  rq_init_comm_if_connected(9, "1")
  rq_init_comm_if_connected(2, "2")
  rq_init_comm_if_connected(3, "3")
  rq_init_comm_if_connected(4, "4")
  rq_print_connected_grippers()
  rq_gripper_communication_thread = run rq_gripper_communication()
  set_closed_norm(100.0, 1)
  set_open_norm(0.0, 1)
  set_closed_mm(0.0, 1)
  set_open_mm(50.0, 1)
  set_closed_norm(100.0, 2)
  set_open_norm(0.0, 2)
  set_closed_mm(0.0, 2)
  set_open_mm(50.0, 2)
  set_closed_norm(100.0, 3)
  set_open_norm(0.0, 3)
  set_closed_mm(0.0, 3)
  set_open_mm(50.0, 3)
  set_closed_norm(100.0, 4)
  set_open_norm(0.0, 4)
  set_closed_mm(0.0, 4)
  set_open_mm(50.0, 4)
  rq_current_limit_enabled = False
  while(not rq_gripper_communication_thread_started):
      sleep(0.008)
  end
  # end: URCap Installation Node
  def ExtractCoinBattery():
    $ 40 "ExtractCoinBattery" "noBreak"
    $ 41 "wp_CoinBatApp≔wp_origin"
    global wp_CoinBatApp=wp_origin
    $ 42 "wp_CoinBatApp[0] = -0.0328"
    wp_CoinBatApp[0] = -0.0328
    $ 43 "wp_CoinBatApp[1] = 0.1238 + 0.002"
    wp_CoinBatApp[1] = 0.1238 + 0.002
    $ 44 "wp_CoinBatApp[2] = 0.07"
    wp_CoinBatApp[2] = 0.07
    $ 45 "MoveL"
    $ 46 "wp_CoinBatApp" "breakAfter"
    movel(pose_trans(Fearure_2_2P_Of, wp_CoinBatApp), a=1.2, v=0.25)
    $ 47 "wp_CoinBatExt≔wp_CoinBatApp"
    global wp_CoinBatExt=wp_CoinBatApp
    $ 48 "wp_CoinBatExt[2] = 0.115"
    wp_CoinBatExt[2] = 0.115
    $ 49 "MoveL"
    $ 50 "wp_CoinBatExt" "breakAfter"
    movel(pose_trans(Fearure_2_2P_Of, wp_CoinBatExt), a=1.2, v=0.25)
    # begin: URCap Program Node
    #   Source: Robotiq_Copilot, 1.22.1.14215, Robotiq Inc.
    #   Type: Find Surface
    $ 51 "Find Surface"
    rq_ft_sensor_disconnected_check()
    rq_zero_sensor()
    sleep(0.1)
    surface_found = rq_linear_search_urcap("X-", 35.000, 0.005000, 0.020000, 1)
    storevar.setvariablepose("rq_findSurface_d2ed8732-a4f1-4f80-aeeb-8b3bdc1d8fba_exitPosition", get_actual_tcp_pose())
    $ 52 "'Add Stop conditions from the Find Surface node'" "noBreak"
    # 'Add Stop conditions from the Find Surface node'
    # end: URCap Program Node
    $ 53 "Wait: 0"
    $ 54 "wp_CoinBatExt[2] = 0.07"
    wp_CoinBatExt[2] = 0.07
    $ 55 "MoveL"
    $ 56 "wp_CoinBatExt" "breakAfter"
    movel(pose_trans(Fearure_2_2P_Of, wp_CoinBatExt), a=1.2, v=0.25)
  end
  def PickPlaceCoinBattery():
    $ 59 "PickPlaceCoinBattery" "noBreak"
    # begin: URCap Program Node
    #   Source: Robotiq_Grippers, 1.8.8.13523, Robotiq Inc.
    #   Type: Gripper
    $ 60 "Gripper Move50% (1)"
    if not(gripper_connected[0]):
      popup("Gripper 1 must be connected to run this program.", "No connection", False, True, True)
    end
    if not(rq_is_gripper_activated("1")):
      popup("Gripper 1 is not activated. Go to Installation tab > Gripper to activate it and run the program again.", "Not activated", False, True, True)
    end
    rq_set_pos_spd_for(128, 255, 0, "1")
    rq_wait_pos_spe_for_request(128, 255, 0, "1")
    rq_go_to("1")
    rq_wait("1")
    # end: URCap Program Node
    $ 61 "wp_PickCoinApp≔wp_origin"
    global wp_PickCoinApp=wp_origin
    $ 62 "wp_PickCoinApp[0] = -0.0328"
    wp_PickCoinApp[0] = -0.0328
    $ 63 "wp_PickCoinApp[1] = 0.1238"
    wp_PickCoinApp[1] = 0.1238
    $ 64 "wp_PickCoinApp[2] = 0.14"
    wp_PickCoinApp[2] = 0.14
    $ 65 "wp_PickCoinApp[5] = d2r(90)"
    wp_PickCoinApp[5] = d2r(90)
    $ 66 "MoveL"
    $ 67 "wp_PickCoinApp" "breakAfter"
    movel(pose_trans(Fearure_2_2P_Of, wp_PickCoinApp), a=1.2, v=0.25)
    # begin: URCap Program Node
    #   Source: Robotiq_Grippers, 1.8.8.13523, Robotiq Inc.
    #   Type: Gripper
    $ 68 "Gripper Close (1)"
    if not(gripper_connected[0]):
      popup("Gripper 1 must be connected to run this program.", "No connection", False, True, True)
    end
    if not(rq_is_gripper_activated("1")):
      popup("Gripper 1 is not activated. Go to Installation tab > Gripper to activate it and run the program again.", "Not activated", False, True, True)
    end
    rq_set_pos_spd_for(255, 0, 0, "1")
    rq_wait_pos_spe_for_request(255, 0, 0, "1")
    rq_go_to("1")
    rq_wait("1")
    # end: URCap Program Node
    $ 69 "wp_PickCoinApp[2] = 0.12"
    wp_PickCoinApp[2] = 0.12
    $ 70 "MoveL"
    $ 71 "wp_PickCoinApp" "breakAfter"
    movel(pose_trans(Fearure_2_2P_Of, wp_PickCoinApp), a=1.2, v=0.25)
    $ 72 "wp_PickCoinApp[1] = 0.09"
    wp_PickCoinApp[1] = 0.09
    $ 73 "MoveL"
    $ 74 "wp_PickCoinApp" "breakAfter"
    movel(pose_trans(Fearure_2_2P_Of, wp_PickCoinApp), a=1.2, v=0.25)
    $ 75 "wp_PickCoinApp[2] = 0.13"
    wp_PickCoinApp[2] = 0.13
    $ 76 "MoveL"
    $ 77 "wp_PickCoinApp" "breakAfter"
    movel(pose_trans(Fearure_2_2P_Of, wp_PickCoinApp), a=1.2, v=0.25)
    # begin: URCap Program Node
    #   Source: Robotiq_Grippers, 1.8.8.13523, Robotiq Inc.
    #   Type: Gripper
    $ 78 "Gripper Move65% (1)"
    if not(gripper_connected[0]):
      popup("Gripper 1 must be connected to run this program.", "No connection", False, True, True)
    end
    if not(rq_is_gripper_activated("1")):
      popup("Gripper 1 is not activated. Go to Installation tab > Gripper to activate it and run the program again.", "Not activated", False, True, True)
    end
    rq_set_pos_spd_for(166, 0, 0, "1")
    rq_wait_pos_spe_for_request(166, 0, 0, "1")
    rq_go_to("1")
    rq_wait("1")
    # end: URCap Program Node
    $ 79 "wp_PickCoinApp[2] = 0"
    wp_PickCoinApp[2] = 0
    $ 80 "MoveL"
    $ 81 "wp_PickCoinApp" "breakAfter"
    movel(pose_trans(Fearure_2_2P_Of, wp_PickCoinApp), a=1.2, v=0.25)
    # begin: URCap Program Node
    #   Source: Robotiq_Grippers, 1.8.8.13523, Robotiq Inc.
    #   Type: Gripper
    $ 82 "Gripper Close (1)"
    if not(gripper_connected[0]):
      popup("Gripper 1 must be connected to run this program.", "No connection", False, True, True)
    end
    if not(rq_is_gripper_activated("1")):
      popup("Gripper 1 is not activated. Go to Installation tab > Gripper to activate it and run the program again.", "Not activated", False, True, True)
    end
    rq_set_pos_spd_for(255, 255, 0, "1")
    rq_wait_pos_spe_for_request(255, 255, 0, "1")
    rq_go_to("1")
    rq_wait("1")
    # end: URCap Program Node
  end
  def ExtractBattery2():
    $ 83 "ExtractBattery2" "noBreak"
    $ 84 "wp_Bat2ExtApp≔wp_origin"
    global wp_Bat2ExtApp=wp_origin
    $ 85 "wp_Bat2ExtApp[0] = -0.10"
    wp_Bat2ExtApp[0] = -0.10
    $ 86 "wp_Bat2ExtApp[1] = 0.06"
    wp_Bat2ExtApp[1] = 0.06
    $ 87 "wp_Bat2ExtApp[2] = 0.07"
    wp_Bat2ExtApp[2] = 0.07
    $ 88 "MoveL"
    $ 89 "wp_Bat2ExtApp" "breakAfter"
    movel(pose_trans(Fearure_2_2P_Of, wp_Bat2ExtApp), a=1.2, v=0.25)
    $ 90 "wp_Bat2ExtApp[2] = 0.115"
    wp_Bat2ExtApp[2] = 0.115
    $ 91 "MoveL"
    $ 92 "wp_Bat2ExtApp" "breakAfter"
    movel(pose_trans(Fearure_2_2P_Of, wp_Bat2ExtApp), a=1.2, v=0.25)
    # begin: URCap Program Node
    #   Source: Robotiq_Copilot, 1.22.1.14215, Robotiq Inc.
    #   Type: Find Surface
    $ 93 "Find Surface"
    rq_ft_sensor_disconnected_check()
    rq_zero_sensor()
    sleep(0.1)
    surface_found = rq_linear_search_urcap("X-", 30.000, 0.020000, 0.030000, 1)
    storevar.setvariablepose("rq_findSurface_fb726c3e-57f5-4e83-bd0d-2e451a65e373_exitPosition", get_actual_tcp_pose())
    $ 94 "'Add Stop conditions from the Find Surface node'" "noBreak"
    # 'Add Stop conditions from the Find Surface node'
    # end: URCap Program Node
    $ 95 "wp_Bat2ExtApp[2] = 0.07"
    wp_Bat2ExtApp[2] = 0.07
    $ 96 "MoveL"
    $ 97 "wp_Bat2ExtApp" "breakAfter"
    movel(pose_trans(Fearure_2_2P_Of, wp_Bat2ExtApp), a=1.2, v=0.25)
  end
  def PickTool():
    $ 98 "PickTool" "noBreak"
    $ 99 "wp_PickToolApp≔wp_CornerOrigin"
    global wp_PickToolApp=wp_CornerOrigin
    $ 100 "wp_PickToolApp[0] = -0.081"
    wp_PickToolApp[0] = -0.081
    $ 101 "wp_PickToolApp[1] = 0.083"
    wp_PickToolApp[1] = 0.083
    $ 102 "MoveL"
    $ 103 "wp_PickToolApp" "breakAfter"
    movel(pose_trans(Fearure_2_2P_Of, wp_PickToolApp), a=1.2, v=0.25)
    # begin: URCap Program Node
    #   Source: Robotiq_Grippers, 1.8.8.13523, Robotiq Inc.
    #   Type: Gripper
    $ 104 "Gripper Move60% (1)"
    if not(gripper_connected[0]):
      popup("Gripper 1 must be connected to run this program.", "No connection", False, True, True)
    end
    if not(rq_is_gripper_activated("1")):
      popup("Gripper 1 is not activated. Go to Installation tab > Gripper to activate it and run the program again.", "Not activated", False, True, True)
    end
    rq_set_pos_spd_for(153, 255, 0, "1")
    rq_wait_pos_spe_for_request(153, 255, 0, "1")
    rq_go_to("1")
    rq_wait("1")
    # end: URCap Program Node
    $ 105 "wp_PickToolApp[2] = 0.148"
    wp_PickToolApp[2] = 0.148
    $ 106 "MoveL"
    $ 107 "wp_PickToolApp" "breakAfter"
    movel(pose_trans(Fearure_2_2P_Of, wp_PickToolApp), a=1.2, v=0.25)
    $ 108 "wp_PickToolApp[1] = 0.08"
    wp_PickToolApp[1] = 0.08
    $ 109 "MoveL"
    $ 110 "wp_PickToolApp" "breakAfter"
    movel(pose_trans(Fearure_2_2P_Of, wp_PickToolApp), a=1.2, v=0.25)
    # begin: URCap Program Node
    #   Source: Robotiq_Grippers, 1.8.8.13523, Robotiq Inc.
    #   Type: Gripper
    $ 111 "Gripper Close (1)"
    if not(gripper_connected[0]):
      popup("Gripper 1 must be connected to run this program.", "No connection", False, True, True)
    end
    if not(rq_is_gripper_activated("1")):
      popup("Gripper 1 is not activated. Go to Installation tab > Gripper to activate it and run the program again.", "Not activated", False, True, True)
    end
    rq_set_pos_spd_for(255, 255, 255, "1")
    rq_wait_pos_spe_for_request(255, 255, 255, "1")
    rq_go_to("1")
    rq_wait("1")
    # end: URCap Program Node
    $ 112 "wp_PickToolApp[2] = 0.07"
    wp_PickToolApp[2] = 0.07
    $ 113 "MoveL"
    $ 114 "wp_PickToolApp" "breakAfter"
    movel(pose_trans(Fearure_2_2P_Of, wp_PickToolApp), a=1.2, v=0.25)
  end
  def PlaceTool():
    $ 115 "PlaceTool" "noBreak"
    $ 116 "wp_PlaceToolApp≔wp_origin"
    global wp_PlaceToolApp=wp_origin
    $ 117 "wp_PlaceToolApp[0] = -0.081"
    wp_PlaceToolApp[0] = -0.081
    $ 118 "wp_PlaceToolApp[1] = 0.08"
    wp_PlaceToolApp[1] = 0.08
    $ 119 "MoveL"
    $ 120 "wp_PlaceToolApp" "breakAfter"
    movel(pose_trans(Fearure_2_2P_Of, wp_PlaceToolApp), a=1.2, v=0.25)
    $ 121 "wp_PlaceToolApp[2] = 0.13"
    wp_PlaceToolApp[2] = 0.13
    $ 122 "MoveL"
    $ 123 "wp_PlaceToolApp" "breakAfter"
    movel(pose_trans(Fearure_2_2P_Of, wp_PlaceToolApp), a=1.2, v=0.25)
    # begin: URCap Program Node
    #   Source: Robotiq_Copilot, 1.22.1.14215, Robotiq Inc.
    #   Type: Insertion
    $ 124 "Insertion"
    rq_ft_sensor_disconnected_check()
    # begin: URCap Program Node
    #   Source: Robotiq_Copilot, 1.22.1.14215, Robotiq Inc.
    #   Type: Zero FT Sensor
    $ 125 "Zero FT Sensor" "noBreak"
    rq_ft_sensor_disconnected_check()
    rq_zero_sensor()
    # end: URCap Program Node
    # begin: URCap Program Node
    #   Source: Robotiq_Copilot, 1.22.1.14215, Robotiq Inc.
    #   Type: Linear
    $ 126 "Linear" "noBreak"
    rq_ft_sensor_disconnected_check()
    surface_found = rq_linear_search_urcap("Z+", 10.000, 0.020, 0.030, 1)
    # begin: URCap Program Node
    #   Source: Robotiq_Copilot, 1.22.1.14215, Robotiq Inc.
    #   Type: On error
    $ 127 "On error" "noBreak"
    if not(surface_found):
      $ 128 "'Sequence if maximum distance is reached'" "noBreak"
      # 'Sequence if maximum distance is reached'
      $ 129 "Halt" "noBreak"
      halt
    end
    # end: URCap Program Node
    # end: URCap Program Node
    # end: URCap Program Node
    # begin: URCap Program Node
    #   Source: Robotiq_Grippers, 1.8.8.13523, Robotiq Inc.
    #   Type: Gripper
    $ 130 "Gripper Move60% (1)"
    if not(gripper_connected[0]):
      popup("Gripper 1 must be connected to run this program.", "No connection", False, True, True)
    end
    if not(rq_is_gripper_activated("1")):
      popup("Gripper 1 is not activated. Go to Installation tab > Gripper to activate it and run the program again.", "Not activated", False, True, True)
    end
    rq_set_pos_spd_for(153, 255, 0, "1")
    rq_wait_pos_spe_for_request(153, 255, 0, "1")
    rq_go_to("1")
    rq_wait("1")
    # end: URCap Program Node
    $ 131 "wp_PlaceToolApp[2] = 0.07"
    wp_PlaceToolApp[2] = 0.07
    $ 132 "MoveL"
    $ 133 "wp_PlaceToolApp" "breakAfter"
    movel(pose_trans(Fearure_2_2P_Of, wp_PlaceToolApp), a=1.2, v=0.25)
    $ 134 "wp_PlaceToolApp[5] = 1.571"
    wp_PlaceToolApp[5] = 1.571
    $ 135 "MoveL"
    $ 136 "wp_PlaceToolApp" "breakAfter"
    movel(pose_trans(Fearure_2_2P_Of, wp_PlaceToolApp), a=1.2, v=0.25)
  end
  def ReleaseTool():
    $ 137 "ReleaseTool" "noBreak"
    $ 138 "wp_RelToolApp≔wp_origin"
    global wp_RelToolApp=wp_origin
    $ 139 "wp_RelToolApp[0] = -0.0328"
    wp_RelToolApp[0] = -0.0328
    $ 140 "wp_RelToolApp[1] = 0.18"
    wp_RelToolApp[1] = 0.18
    $ 141 "wp_RelToolApp[2] = 0.07"
    wp_RelToolApp[2] = 0.07
    $ 142 "MoveL"
    $ 143 "wp_RelToolApp" "breakAfter"
    movel(pose_trans(Fearure_2_2P_Of, wp_RelToolApp), a=1.2, v=0.25)
    # begin: URCap Program Node
    #   Source: Robotiq_Grippers, 1.8.8.13523, Robotiq Inc.
    #   Type: Gripper
    $ 144 "Gripper Move50% (1)"
    if not(gripper_connected[0]):
      popup("Gripper 1 must be connected to run this program.", "No connection", False, True, True)
    end
    if not(rq_is_gripper_activated("1")):
      popup("Gripper 1 is not activated. Go to Installation tab > Gripper to activate it and run the program again.", "Not activated", False, True, True)
    end
    rq_set_pos_spd_for(128, 255, 0, "1")
    rq_wait_pos_spe_for_request(128, 255, 0, "1")
    rq_go_to("1")
    rq_wait("1")
    # end: URCap Program Node
    $ 145 "wp_RelToolApp[2] = 0"
    wp_RelToolApp[2] = 0
    $ 146 "MoveL"
    $ 147 "wp_RelToolApp" "breakAfter"
    movel(pose_trans(Fearure_2_2P_Of, wp_RelToolApp), a=1.2, v=0.25)
    # begin: URCap Program Node
    #   Source: Robotiq_Grippers, 1.8.8.13523, Robotiq Inc.
    #   Type: Gripper
    $ 148 "Gripper Close (1)"
    if not(gripper_connected[0]):
      popup("Gripper 1 must be connected to run this program.", "No connection", False, True, True)
    end
    if not(rq_is_gripper_activated("1")):
      popup("Gripper 1 is not activated. Go to Installation tab > Gripper to activate it and run the program again.", "Not activated", False, True, True)
    end
    rq_set_pos_spd_for(255, 255, 0, "1")
    rq_wait_pos_spe_for_request(255, 255, 0, "1")
    rq_go_to("1")
    rq_wait("1")
    # end: URCap Program Node
  end
  def InsertBattery1():
    $ 149 "InsertBattery1" "noBreak"
    $ 150 "wp_InsBat1App≔wp_origin"
    global wp_InsBat1App=wp_origin
    $ 151 "wp_InsBat1App[0] = wp_InsBat1App[0] - 0.042"
    wp_InsBat1App[0] = wp_InsBat1App[0] - 0.042
    $ 152 "wp_InsBat1App[1] = wp_InsBat1App[1] + 0.0555"
    wp_InsBat1App[1] = wp_InsBat1App[1] + 0.0555
    $ 153 "MoveL"
    $ 154 "wp_InsBat1App" "breakAfter"
    movel(pose_trans(Fearure_2_2P_Of, wp_InsBat1App), a=1.2, v=0.25)
    $ 156 "wp_InsBat1App[2] = wp_InsBat1App[2] + 0.08"
    wp_InsBat1App[2] = wp_InsBat1App[2] + 0.08
    $ 157 "wp_InsBat1App[0] = wp_InsBat1App[0] + 0.005"
    wp_InsBat1App[0] = wp_InsBat1App[0] + 0.005
    $ 158 "MoveL"
    $ 159 "wp_InsBat1App" "breakAfter"
    movel(pose_trans(Fearure_2_2P_Of, wp_InsBat1App), a=1.2, v=0.25)
    # begin: URCap Program Node
    #   Source: Robotiq_Copilot, 1.22.1.14215, Robotiq Inc.
    #   Type: Insertion
    $ 160 "Insertion"
    rq_ft_sensor_disconnected_check()
    # begin: URCap Program Node
    #   Source: Robotiq_Copilot, 1.22.1.14215, Robotiq Inc.
    #   Type: Zero FT Sensor
    $ 161 "Zero FT Sensor" "noBreak"
    rq_ft_sensor_disconnected_check()
    rq_zero_sensor()
    # end: URCap Program Node
    # begin: URCap Program Node
    #   Source: Robotiq_Copilot, 1.22.1.14215, Robotiq Inc.
    #   Type: Linear
    $ 162 "Linear" "noBreak"
    rq_ft_sensor_disconnected_check()
    surface_found = rq_linear_search_urcap("Z+", 10.000, 0.010, 0.030, 1)
    # begin: URCap Program Node
    #   Source: Robotiq_Copilot, 1.22.1.14215, Robotiq Inc.
    #   Type: On error
    $ 163 "On error" "noBreak"
    if not(surface_found):
      $ 164 "'Sequence if maximum distance is reached'" "noBreak"
      # 'Sequence if maximum distance is reached'
      $ 165 "Halt" "noBreak"
      halt
    end
    # end: URCap Program Node
    # end: URCap Program Node
    # end: URCap Program Node
    $ 166 "Wait: 0.5"
    sleep(0.5)
    # begin: URCap Program Node
    #   Source: Robotiq_Grippers, 1.8.8.13523, Robotiq Inc.
    #   Type: Gripper
    $ 167 "Gripper Move60% (1)"
    if not(gripper_connected[0]):
      popup("Gripper 1 must be connected to run this program.", "No connection", False, True, True)
    end
    if not(rq_is_gripper_activated("1")):
      popup("Gripper 1 is not activated. Go to Installation tab > Gripper to activate it and run the program again.", "Not activated", False, True, True)
    end
    rq_set_pos_spd_for(153, 255, 0, "1")
    rq_wait_pos_spe_for_request(153, 255, 0, "1")
    rq_go_to("1")
    rq_wait("1")
    # end: URCap Program Node
    $ 168 "wp_InsBat1Ret≔wp_InsBat1App"
    global wp_InsBat1Ret=wp_InsBat1App
    $ 169 "wp_InsBat1Ret[2] = wp_InsBat1Ret[2] - 0.10"
    wp_InsBat1Ret[2] = wp_InsBat1Ret[2] - 0.10
    $ 170 "MoveL"
    $ 171 "wp_InsBat1Ret" "breakAfter"
    movel(pose_trans(Fearure_2_2P_Of, wp_InsBat1Ret), a=1.2, v=0.25)
    # begin: URCap Program Node
    #   Source: Robotiq_Grippers, 1.8.8.13523, Robotiq Inc.
    #   Type: Gripper
    $ 172 "Gripper Close (1)"
    if not(gripper_connected[0]):
      popup("Gripper 1 must be connected to run this program.", "No connection", False, True, True)
    end
    if not(rq_is_gripper_activated("1")):
      popup("Gripper 1 is not activated. Go to Installation tab > Gripper to activate it and run the program again.", "Not activated", False, True, True)
    end
    rq_set_pos_spd_for(255, 255, 0, "1")
    rq_wait_pos_spe_for_request(255, 255, 0, "1")
    rq_go_to("1")
    rq_wait("1")
    # end: URCap Program Node
  end
  def InsertBattery2():
    $ 179 "InsertBattery2" "noBreak"
    $ 180 "wp_InsBat2App≔wp_origin"
    global wp_InsBat2App=wp_origin
    $ 181 "wp_InsBat2App[0] = -0.058"
    wp_InsBat2App[0] = -0.058
    $ 182 "wp_InsBat2App[1] = 0.0555"
    wp_InsBat2App[1] = 0.0555
    $ 183 "wp_InsBat2App[5] = 1.571"
    wp_InsBat2App[5] = 1.571
    $ 184 "MoveL"
    $ 185 "wp_InsBat2App" "breakAfter"
    movel(pose_trans(Fearure_2_2P_Of, wp_InsBat2App), a=1.2, v=0.25)
    $ 186 "wp_InsBat2App[2] = 0.08"
    wp_InsBat2App[2] = 0.08
    $ 187 "wp_InsBat2App[0] = wp_InsBat2App[0] - 0.005"
    wp_InsBat2App[0] = wp_InsBat2App[0] - 0.005
    $ 188 "MoveL"
    $ 189 "wp_InsBat2App" "breakAfter"
    movel(pose_trans(Fearure_2_2P_Of, wp_InsBat2App), a=1.2, v=0.25)
    # begin: URCap Program Node
    #   Source: Robotiq_Copilot, 1.22.1.14215, Robotiq Inc.
    #   Type: Insertion
    $ 190 "Insertion"
    rq_ft_sensor_disconnected_check()
    # begin: URCap Program Node
    #   Source: Robotiq_Copilot, 1.22.1.14215, Robotiq Inc.
    #   Type: Zero FT Sensor
    $ 191 "Zero FT Sensor" "noBreak"
    rq_ft_sensor_disconnected_check()
    rq_zero_sensor()
    # end: URCap Program Node
    # begin: URCap Program Node
    #   Source: Robotiq_Copilot, 1.22.1.14215, Robotiq Inc.
    #   Type: Linear
    $ 192 "Linear" "noBreak"
    rq_ft_sensor_disconnected_check()
    surface_found = rq_linear_search_urcap("Z+", 10.000, 0.010, 0.030, 1)
    # begin: URCap Program Node
    #   Source: Robotiq_Copilot, 1.22.1.14215, Robotiq Inc.
    #   Type: On error
    $ 193 "On error" "noBreak"
    if not(surface_found):
      $ 194 "'Sequence if maximum distance is reached'" "noBreak"
      # 'Sequence if maximum distance is reached'
      $ 195 "Halt" "noBreak"
      halt
    end
    # end: URCap Program Node
    # end: URCap Program Node
    # end: URCap Program Node
    $ 196 "Wait: 0.5"
    sleep(0.5)
    # begin: URCap Program Node
    #   Source: Robotiq_Grippers, 1.8.8.13523, Robotiq Inc.
    #   Type: Gripper
    $ 197 "Gripper Move60% (1)"
    if not(gripper_connected[0]):
      popup("Gripper 1 must be connected to run this program.", "No connection", False, True, True)
    end
    if not(rq_is_gripper_activated("1")):
      popup("Gripper 1 is not activated. Go to Installation tab > Gripper to activate it and run the program again.", "Not activated", False, True, True)
    end
    rq_set_pos_spd_for(153, 255, 0, "1")
    rq_wait_pos_spe_for_request(153, 255, 0, "1")
    rq_go_to("1")
    rq_wait("1")
    # end: URCap Program Node
    $ 198 "wp_InsBat2Ret≔wp_InsBat2App"
    global wp_InsBat2Ret=wp_InsBat2App
    $ 199 "wp_InsBat2Ret[2] = wp_InsBat2Ret[2] - 0.10"
    wp_InsBat2Ret[2] = wp_InsBat2Ret[2] - 0.10
    $ 200 "MoveL"
    $ 201 "wp_InsBat2Ret" "breakAfter"
    movel(pose_trans(Fearure_2_2P_Of, wp_InsBat2Ret), a=1.2, v=0.25)
    # begin: URCap Program Node
    #   Source: Robotiq_Grippers, 1.8.8.13523, Robotiq Inc.
    #   Type: Gripper
    $ 202 "Gripper Close (1)"
    if not(gripper_connected[0]):
      popup("Gripper 1 must be connected to run this program.", "No connection", False, True, True)
    end
    if not(rq_is_gripper_activated("1")):
      popup("Gripper 1 is not activated. Go to Installation tab > Gripper to activate it and run the program again.", "Not activated", False, True, True)
    end
    rq_set_pos_spd_for(255, 255, 0, "1")
    rq_wait_pos_spe_for_request(255, 255, 0, "1")
    rq_go_to("1")
    rq_wait("1")
    # end: URCap Program Node
  end
  def PickBattery2():
    $ 203 "PickBattery2" "noBreak"
    # begin: URCap Program Node
    #   Source: Robotiq_Grippers, 1.8.8.13523, Robotiq Inc.
    #   Type: Gripper
    $ 204 "Gripper Move60% (1)"
    if not(gripper_connected[0]):
      popup("Gripper 1 must be connected to run this program.", "No connection", False, True, True)
    end
    if not(rq_is_gripper_activated("1")):
      popup("Gripper 1 is not activated. Go to Installation tab > Gripper to activate it and run the program again.", "Not activated", False, True, True)
    end
    rq_set_pos_spd_for(153, 0, 0, "1")
    rq_wait_pos_spe_for_request(153, 0, 0, "1")
    rq_go_to("1")
    rq_wait("1")
    # end: URCap Program Node
    $ 205 "wp_Bat2PickApp≔wp_origin"
    global wp_Bat2PickApp=wp_origin
    $ 206 "wp_Bat2PickApp[0] = -0.1045"
    wp_Bat2PickApp[0] = -0.1045
    $ 207 "wp_Bat2PickApp[1] = 0.0565"
    wp_Bat2PickApp[1] = 0.0565
    $ 208 "wp_Bat2PickApp[5] = 1.571"
    wp_Bat2PickApp[5] = 1.571
    $ 209 "MoveL"
    $ 210 "wp_Bat2PickApp" "breakAfter"
    movel(pose_trans(Fearure_2_2P_Of, wp_Bat2PickApp), a=1.2, v=0.25)
    $ 211 "wp_Bat2PickApp[2] = 0.134"
    wp_Bat2PickApp[2] = 0.134
    $ 212 "MoveL"
    $ 213 "wp_Bat2PickApp" "breakAfter"
    movel(pose_trans(Fearure_2_2P_Of, wp_Bat2PickApp), a=1.2, v=0.25)
    # begin: URCap Program Node
    #   Source: Robotiq_Grippers, 1.8.8.13523, Robotiq Inc.
    #   Type: Gripper
    $ 214 "Gripper Close (1)"
    if not(gripper_connected[0]):
      popup("Gripper 1 must be connected to run this program.", "No connection", False, True, True)
    end
    if not(rq_is_gripper_activated("1")):
      popup("Gripper 1 is not activated. Go to Installation tab > Gripper to activate it and run the program again.", "Not activated", False, True, True)
    end
    rq_set_pos_spd_for(255, 128, 0, "1")
    rq_wait_pos_spe_for_request(255, 128, 0, "1")
    rq_go_to("1")
    rq_wait("1")
    # end: URCap Program Node
    $ 215 "wp_Bat2PickApp[2] = 0.07"
    wp_Bat2PickApp[2] = 0.07
    $ 216 "MoveL"
    $ 217 "wp_Bat2PickApp" "breakAfter"
    movel(pose_trans(Fearure_2_2P_Of, wp_Bat2PickApp), a=1.2, v=0.25)
    # begin: URCap Program Node
    #   Source: Robotiq_Grippers, 1.8.8.13523, Robotiq Inc.
    #   Type: Gripper
    $ 218 "Gripper Move72% (1)"
    if not(gripper_connected[0]):
      popup("Gripper 1 must be connected to run this program.", "No connection", False, True, True)
    end
    if not(rq_is_gripper_activated("1")):
      popup("Gripper 1 is not activated. Go to Installation tab > Gripper to activate it and run the program again.", "Not activated", False, True, True)
    end
    rq_set_pos_spd_for(184, 0, 0, "1")
    rq_wait_pos_spe_for_request(184, 0, 0, "1")
    rq_go_to("1")
    rq_wait("1")
    # end: URCap Program Node
    $ 219 "Wait: 3.0"
    sleep(3.0)
    # begin: URCap Program Node
    #   Source: Robotiq_Grippers, 1.8.8.13523, Robotiq Inc.
    #   Type: Gripper
    $ 220 "Gripper Move85% (1)"
    if not(gripper_connected[0]):
      popup("Gripper 1 must be connected to run this program.", "No connection", False, True, True)
    end
    if not(rq_is_gripper_activated("1")):
      popup("Gripper 1 is not activated. Go to Installation tab > Gripper to activate it and run the program again.", "Not activated", False, True, True)
    end
    rq_set_pos_spd_for(217, 255, 0, "1")
    rq_wait_pos_spe_for_request(217, 255, 0, "1")
    rq_go_to("1")
    rq_wait("1")
    # end: URCap Program Node
  end
  def PickBattery1():
    $ 221 "PickBattery1" "noBreak"
    # begin: URCap Program Node
    #   Source: Robotiq_Grippers, 1.8.8.13523, Robotiq Inc.
    #   Type: Gripper
    $ 222 "Gripper Move60% (1)"
    if not(gripper_connected[0]):
      popup("Gripper 1 must be connected to run this program.", "No connection", False, True, True)
    end
    if not(rq_is_gripper_activated("1")):
      popup("Gripper 1 is not activated. Go to Installation tab > Gripper to activate it and run the program again.", "Not activated", False, True, True)
    end
    rq_set_pos_spd_for(153, 0, 0, "1")
    rq_wait_pos_spe_for_request(153, 0, 0, "1")
    rq_go_to("1")
    rq_wait("1")
    # end: URCap Program Node
    $ 223 "wp_Bat1ExtApp≔wp_origin"
    global wp_Bat1ExtApp=wp_origin
    $ 224 "wp_Bat1ExtApp[0] = wp_Bat1ExtApp[0] - 0.1540"
    wp_Bat1ExtApp[0] = wp_Bat1ExtApp[0] - 0.1540
    $ 225 "wp_Bat1ExtApp[1] = wp_Bat1ExtApp[1] + 0.0415"
    wp_Bat1ExtApp[1] = wp_Bat1ExtApp[1] + 0.0415
    $ 226 "wp_Bat1ExtApp[5] = wp_Bat1ExtApp[5] + 1.571"
    wp_Bat1ExtApp[5] = wp_Bat1ExtApp[5] + 1.571
    $ 227 "MoveL"
    $ 228 "wp_Bat1ExtApp" "breakAfter"
    movel(pose_trans(Fearure_2_2P_Of, wp_Bat1ExtApp), a=1.2, v=0.25)
    $ 229 "wp_Bat1ExtApp[2] = wp_Bat1ExtApp[2] + 0.136"
    wp_Bat1ExtApp[2] = wp_Bat1ExtApp[2] + 0.136
    $ 230 "MoveL"
    $ 231 "wp_Bat1ExtApp" "breakAfter"
    movel(pose_trans(Fearure_2_2P_Of, wp_Bat1ExtApp), a=1.2, v=0.25)
    # begin: URCap Program Node
    #   Source: Robotiq_Grippers, 1.8.8.13523, Robotiq Inc.
    #   Type: Gripper
    $ 232 "Gripper Close (1)"
    if not(gripper_connected[0]):
      popup("Gripper 1 must be connected to run this program.", "No connection", False, True, True)
    end
    if not(rq_is_gripper_activated("1")):
      popup("Gripper 1 is not activated. Go to Installation tab > Gripper to activate it and run the program again.", "Not activated", False, True, True)
    end
    rq_set_pos_spd_for(255, 0, 0, "1")
    rq_wait_pos_spe_for_request(255, 0, 0, "1")
    rq_go_to("1")
    rq_wait("1")
    # end: URCap Program Node
    $ 233 "wp_Bat1ExtApp[2] = wp_Bat1ExtApp[2] - 0.10"
    wp_Bat1ExtApp[2] = wp_Bat1ExtApp[2] - 0.10
    $ 234 "MoveL"
    $ 235 "wp_Bat1ExtApp" "breakAfter"
    movel(pose_trans(Fearure_2_2P_Of, wp_Bat1ExtApp), a=1.2, v=0.25)
    # begin: URCap Program Node
    #   Source: Robotiq_Grippers, 1.8.8.13523, Robotiq Inc.
    #   Type: Gripper
    $ 236 "Gripper Move72% (1)"
    if not(gripper_connected[0]):
      popup("Gripper 1 must be connected to run this program.", "No connection", False, True, True)
    end
    if not(rq_is_gripper_activated("1")):
      popup("Gripper 1 is not activated. Go to Installation tab > Gripper to activate it and run the program again.", "Not activated", False, True, True)
    end
    rq_set_pos_spd_for(184, 0, 0, "1")
    rq_wait_pos_spe_for_request(184, 0, 0, "1")
    rq_go_to("1")
    rq_wait("1")
    # end: URCap Program Node
    $ 237 "Wait: 3.0"
    sleep(3.0)
    # begin: URCap Program Node
    #   Source: Robotiq_Grippers, 1.8.8.13523, Robotiq Inc.
    #   Type: Gripper
    $ 238 "Gripper Move85% (1)"
    if not(gripper_connected[0]):
      popup("Gripper 1 must be connected to run this program.", "No connection", False, True, True)
    end
    if not(rq_is_gripper_activated("1")):
      popup("Gripper 1 is not activated. Go to Installation tab > Gripper to activate it and run the program again.", "Not activated", False, True, True)
    end
    rq_set_pos_spd_for(217, 255, 0, "1")
    rq_wait_pos_spe_for_request(217, 255, 0, "1")
    rq_go_to("1")
    rq_wait("1")
    # end: URCap Program Node
  end
  def ExtractBattery1():
    $ 239 "ExtractBattery1" "noBreak"
    $ 240 "wp_Bat1ExtApp≔wp_origin"
    global wp_Bat1ExtApp=wp_origin
    $ 241 "wp_Bat1ExtApp[0] = wp_Bat1ExtApp[0] - 0.1540"
    wp_Bat1ExtApp[0] = wp_Bat1ExtApp[0] - 0.1540
    $ 242 "wp_Bat1ExtApp[1] = wp_Bat1ExtApp[1] + 0.0415"
    wp_Bat1ExtApp[1] = wp_Bat1ExtApp[1] + 0.0415
    $ 243 "MoveL"
    $ 244 "wp_Bat1ExtApp" "breakAfter"
    movel(pose_trans(Fearure_2_2P_Of, wp_Bat1ExtApp), a=1.2, v=0.25)
    # begin: URCap Program Node
    #   Source: Robotiq_Grippers, 1.8.8.13523, Robotiq Inc.
    #   Type: Gripper
    $ 245 "Gripper Move30% (1)"
    if not(gripper_connected[0]):
      popup("Gripper 1 must be connected to run this program.", "No connection", False, True, True)
    end
    if not(rq_is_gripper_activated("1")):
      popup("Gripper 1 is not activated. Go to Installation tab > Gripper to activate it and run the program again.", "Not activated", False, True, True)
    end
    rq_set_pos_spd_for(77, 0, 0, "1")
    rq_wait_pos_spe_for_request(77, 0, 0, "1")
    rq_go_to("1")
    rq_wait("1")
    # end: URCap Program Node
    $ 246 "wp_Bat1Extract≔wp_Bat1ExtApp"
    global wp_Bat1Extract=wp_Bat1ExtApp
    $ 247 "wp_Bat1Extract[0] = wp_Bat1Extract[0] + 0.034"
    wp_Bat1Extract[0] = wp_Bat1Extract[0] + 0.034
    $ 248 "wp_Bat1Extract[1] = wp_Bat1Extract[1] - 0.01"
    wp_Bat1Extract[1] = wp_Bat1Extract[1] - 0.01
    $ 249 "wp_Bat1Extract[2] = wp_Bat1Extract[2] + 0.145"
    wp_Bat1Extract[2] = wp_Bat1Extract[2] + 0.145
    $ 250 "MoveL"
    $ 251 "wp_Bat1Extract" "breakAfter"
    movel(pose_trans(Fearure_2_2P_Of, wp_Bat1Extract), a=1.2, v=0.25)
    # begin: URCap Program Node
    #   Source: Robotiq_Copilot, 1.22.1.14215, Robotiq Inc.
    #   Type: Find Surface
    $ 252 "Find Surface"
    rq_ft_sensor_disconnected_check()
    rq_zero_sensor()
    sleep(0.1)
    surface_found = rq_linear_search_urcap("X+", 30.000, 0.030000, 0.010000, 1)
    storevar.setvariablepose("rq_findSurface_26ca67e9-cc0e-4d30-826d-8f6b0826683b_exitPosition", get_actual_tcp_pose())
    $ 253 "'Add Stop conditions from the Find Surface node'" "noBreak"
    # 'Add Stop conditions from the Find Surface node'
    # end: URCap Program Node
    $ 254 "wp_Bat1Extract[2] = wp_Bat1Extract[2] - 0.05"
    wp_Bat1Extract[2] = wp_Bat1Extract[2] - 0.05
    $ 255 "MoveL"
    $ 256 "wp_Bat1Extract" "breakAfter"
    movel(pose_trans(Fearure_2_2P_Of, wp_Bat1Extract), a=1.2, v=0.5)
    # begin: URCap Program Node
    #   Source: Robotiq_Grippers, 1.8.8.13523, Robotiq Inc.
    #   Type: Gripper
    $ 257 "Gripper Move60% (1)"
    if not(gripper_connected[0]):
      popup("Gripper 1 must be connected to run this program.", "No connection", False, True, True)
    end
    if not(rq_is_gripper_activated("1")):
      popup("Gripper 1 is not activated. Go to Installation tab > Gripper to activate it and run the program again.", "Not activated", False, True, True)
    end
    rq_set_pos_spd_for(153, 0, 0, "1")
    rq_wait_pos_spe_for_request(153, 0, 0, "1")
    rq_go_to("1")
    rq_wait("1")
    # end: URCap Program Node
  end
  def AABatteryCoverExtraction():
    $ 258 "AABatteryCoverExtraction" "noBreak"
    $ 259 "wp_AABatCovApp≔wp_origin"
    global wp_AABatCovApp=wp_origin
    $ 260 "wp_AABatCovApp[0] = wp_AABatCovApp[0] - 0.1125"
    wp_AABatCovApp[0] = wp_AABatCovApp[0] - 0.1125
    $ 261 "wp_AABatCovApp[1] = wp_AABatCovApp[1] + 0.0485"
    wp_AABatCovApp[1] = wp_AABatCovApp[1] + 0.0485
    $ 262 "MoveL"
    $ 263 "wp_AABatCovApp" "breakAfter"
    movel(pose_trans(Fearure_2_2P_Of, wp_AABatCovApp), a=1.2, v=0.25)
    $ 264 "wp_AABatCovPres≔wp_AABatCovApp"
    global wp_AABatCovPres=wp_AABatCovApp
    $ 265 "wp_AABatCovPres[3] = wp_AABatCovPres[3] + 0.7854"
    wp_AABatCovPres[3] = wp_AABatCovPres[3] + 0.7854
    $ 266 "wp_AABatCovPres[2] = wp_AABatCovPres[2] + 0.12"
    wp_AABatCovPres[2] = wp_AABatCovPres[2] + 0.12
    $ 267 "wp_AABatCovPres[1] = wp_AABatCovPres[1] - 0.008"
    wp_AABatCovPres[1] = wp_AABatCovPres[1] - 0.008
    $ 268 "wp_AABatCovPres[0] = wp_AABatCovPres[0] + 0.005"
    wp_AABatCovPres[0] = wp_AABatCovPres[0] + 0.005
    $ 269 "MoveL"
    $ 270 "wp_AABatCovPres" "breakAfter"
    movel(pose_trans(Fearure_2_2P_Of, wp_AABatCovPres), a=1.2, v=0.25)
    # begin: URCap Program Node
    #   Source: Robotiq_Copilot, 1.22.1.14215, Robotiq Inc.
    #   Type: Find Surface
    $ 271 "Find Surface"
    rq_ft_sensor_disconnected_check()
    rq_zero_sensor()
    sleep(0.1)
    surface_found = rq_linear_search_urcap("Z-", 15.000, 0.030000, 0.010000, 0)
    storevar.setvariablepose("rq_findSurface_54677085-d0b4-4075-8ce2-dc145cac5c67_exitPosition", get_actual_tcp_pose())
    $ 272 "'Add Stop conditions from the Find Surface node'" "noBreak"
    # 'Add Stop conditions from the Find Surface node'
    # end: URCap Program Node
    $ 273 "wp_AABatCovRem≔wp_AABatCovPres"
    global wp_AABatCovRem=wp_AABatCovPres
    $ 274 "wp_AABatCovRem[2] = wp_AABatCovRem[2] + 0.009"
    wp_AABatCovRem[2] = wp_AABatCovRem[2] + 0.009
    $ 275 "wp_AABatCovRem[0] = wp_AABatCovRem[0] - 0.07"
    wp_AABatCovRem[0] = wp_AABatCovRem[0] - 0.07
    $ 276 "MoveL"
    $ 277 "wp_AABatCovRem" "breakAfter"
    movel(pose_trans(Fearure_2_2P_Of, wp_AABatCovRem), a=1.2, v=0.25)
  end
  def PlugInsertion():
    $ 294 "PlugInsertion" "noBreak"
    $ 295 "wp_PlgInsApp≔wp_origin"
    global wp_PlgInsApp=wp_origin
    $ 296 "wp_PlgInsApp[0] =wp_PlgInsApp[0] - 0.1390"
    wp_PlgInsApp[0] =wp_PlgInsApp[0] - 0.1390
    $ 297 "wp_PlgInsApp[1] =wp_PlgInsApp[1] + 0.1065"
    wp_PlgInsApp[1] =wp_PlgInsApp[1] + 0.1065
    $ 298 "wp_PlgInsApp[2] =wp_PlgInsApp[2] + 0.1085"
    wp_PlgInsApp[2] =wp_PlgInsApp[2] + 0.1085
    $ 299 "wp_PlgInsApp[5] = 1.571"
    wp_PlgInsApp[5] = 1.571
    $ 300 "MoveL"
    $ 301 "wp_PlgInsApp" "breakAfter"
    movel(pose_trans(Fearure_2_2P_Of, wp_PlgInsApp), a=1.2, v=0.25)
    $ 302 "wp_PlgInsertion≔wp_PlgInsApp"
    global wp_PlgInsertion=wp_PlgInsApp
    $ 303 "wp_PlgInsertion[2] = wp_PlgInsertion[2] + 0.025"
    wp_PlgInsertion[2] = wp_PlgInsertion[2] + 0.025
    $ 304 "MoveL"
    $ 305 "wp_PlgInsertion" "breakAfter"
    movel(pose_trans(Fearure_2_2P_Of, wp_PlgInsertion), a=1.2, v=0.25)
    # begin: URCap Program Node
    #   Source: Robotiq_Copilot, 1.22.1.14215, Robotiq Inc.
    #   Type: Insertion
    $ 306 "Insertion"
    rq_ft_sensor_disconnected_check()
    # begin: URCap Program Node
    #   Source: Robotiq_Copilot, 1.22.1.14215, Robotiq Inc.
    #   Type: Zero FT Sensor
    $ 307 "Zero FT Sensor" "noBreak"
    rq_ft_sensor_disconnected_check()
    rq_zero_sensor()
    # end: URCap Program Node
    # begin: URCap Program Node
    #   Source: Robotiq_Copilot, 1.22.1.14215, Robotiq Inc.
    #   Type: Linear
    $ 308 "Linear" "noBreak"
    rq_ft_sensor_disconnected_check()
    surface_found = rq_linear_search_urcap("Z+", 10.000, 0.010, 0.015, 1)
    # begin: URCap Program Node
    #   Source: Robotiq_Copilot, 1.22.1.14215, Robotiq Inc.
    #   Type: On error
    $ 309 "On error" "noBreak"
    if not(surface_found):
      $ 310 "'Sequence if maximum distance is reached'" "noBreak"
      # 'Sequence if maximum distance is reached'
      $ 311 "Halt" "noBreak"
      halt
    end
    # end: URCap Program Node
    # end: URCap Program Node
    # end: URCap Program Node
    # begin: URCap Program Node
    #   Source: Robotiq_Grippers, 1.8.8.13523, Robotiq Inc.
    #   Type: Gripper
    $ 312 "Gripper Move60% (1)"
    if not(gripper_connected[0]):
      popup("Gripper 1 must be connected to run this program.", "No connection", False, True, True)
    end
    if not(rq_is_gripper_activated("1")):
      popup("Gripper 1 is not activated. Go to Installation tab > Gripper to activate it and run the program again.", "Not activated", False, True, True)
    end
    rq_set_pos_spd_for(153, 128, 0, "1")
    rq_wait_pos_spe_for_request(153, 128, 0, "1")
    rq_go_to("1")
    rq_wait("1")
    # end: URCap Program Node
    $ 313 "wp_PlgInsRet≔wp_PlgInsertion"
    global wp_PlgInsRet=wp_PlgInsertion
    $ 314 "wp_PlgInsRet[2] = wp_PlgInsRet[2] - 0.1485"
    wp_PlgInsRet[2] = wp_PlgInsRet[2] - 0.1485
    $ 315 "MoveL"
    $ 316 "wp_PlgInsRet" "breakAfter"
    movel(pose_trans(Fearure_2_2P_Of, wp_PlgInsRet), a=1.2, v=0.25)
    # begin: URCap Program Node
    #   Source: Robotiq_Grippers, 1.8.8.13523, Robotiq Inc.
    #   Type: Gripper
    $ 317 "Gripper Close (1)"
    if not(gripper_connected[0]):
      popup("Gripper 1 must be connected to run this program.", "No connection", False, True, True)
    end
    if not(rq_is_gripper_activated("1")):
      popup("Gripper 1 is not activated. Go to Installation tab > Gripper to activate it and run the program again.", "Not activated", False, True, True)
    end
    rq_set_pos_spd_for(255, 128, 0, "1")
    rq_wait_pos_spe_for_request(255, 128, 0, "1")
    rq_go_to("1")
    rq_wait("1")
    # end: URCap Program Node
    $ 318 "wp_PlgInsRet[5] = 0"
    wp_PlgInsRet[5] = 0
    $ 319 "MoveL"
    $ 320 "wp_PlgInsRet" "breakAfter"
    movel(pose_trans(Fearure_2_2P_Of, wp_PlgInsRet), a=1.2, v=0.25)
  end
  def PlugExtraction():
    $ 321 "PlugExtraction" "noBreak"
    $ 322 "wp_PlgExtApp≔wp_origin"
    global wp_PlgExtApp=wp_origin
    $ 323 "wp_PlgExtApp[0] = wp_PlgExtApp[0] - 0.0990"
    wp_PlgExtApp[0] = wp_PlgExtApp[0] - 0.0990
    $ 324 "wp_PlgExtApp[1] = wp_PlgExtApp[1] + 0.1075"
    wp_PlgExtApp[1] = wp_PlgExtApp[1] + 0.1075
    $ 325 "wp_PlgExtApp[5] = 1.571"
    wp_PlgExtApp[5] = 1.571
    $ 326 "MoveL"
    $ 327 "wp_PlgExtApp" "breakAfter"
    movel(pose_trans(Fearure_2_2P_Of, wp_PlgExtApp), a=1.2, v=0.25)
    # begin: URCap Program Node
    #   Source: Robotiq_Grippers, 1.8.8.13523, Robotiq Inc.
    #   Type: Gripper
    $ 328 "Gripper Move60% (1)"
    if not(gripper_connected[0]):
      popup("Gripper 1 must be connected to run this program.", "No connection", False, True, True)
    end
    if not(rq_is_gripper_activated("1")):
      popup("Gripper 1 is not activated. Go to Installation tab > Gripper to activate it and run the program again.", "Not activated", False, True, True)
    end
    rq_set_pos_spd_for(153, 0, 0, "1")
    rq_wait_pos_spe_for_request(153, 0, 0, "1")
    rq_go_to("1")
    rq_wait("1")
    # end: URCap Program Node
    $ 329 "wp_PlgExtract≔wp_PlgExtApp"
    global wp_PlgExtract=wp_PlgExtApp
    $ 330 "wp_PlgExtract[2] = wp_PlgExtract[2] + 0.1385"
    wp_PlgExtract[2] = wp_PlgExtract[2] + 0.1385
    $ 331 "MoveL"
    $ 332 "wp_PlgExtract" "breakAfter"
    movel(pose_trans(Fearure_2_2P_Of, wp_PlgExtract), a=1.2, v=0.25)
    # begin: URCap Program Node
    #   Source: Robotiq_Grippers, 1.8.8.13523, Robotiq Inc.
    #   Type: Gripper
    $ 333 "Gripper Close (1)"
    if not(gripper_connected[0]):
      popup("Gripper 1 must be connected to run this program.", "No connection", False, True, True)
    end
    if not(rq_is_gripper_activated("1")):
      popup("Gripper 1 is not activated. Go to Installation tab > Gripper to activate it and run the program again.", "Not activated", False, True, True)
    end
    rq_set_pos_spd_for(255, 0, 255, "1")
    rq_wait_pos_spe_for_request(255, 0, 255, "1")
    rq_go_to("1")
    rq_wait("1")
    # end: URCap Program Node
    $ 334 "wp_PlgExtRet≔wp_PlgExtract"
    global wp_PlgExtRet=wp_PlgExtract
    $ 335 "wp_PlgExtRet[2] = wp_PlgExtRet[2] - 0.03"
    wp_PlgExtRet[2] = wp_PlgExtRet[2] - 0.03
    $ 336 "MoveL"
    $ 337 "wp_PlgExtRet" "breakAfter"
    movel(pose_trans(Fearure_2_2P_Of, wp_PlgExtRet), a=1.2, v=0.25)
  end
  def KeyInsertion():
    $ 338 "KeyInsertion" "noBreak"
    $ 339 "wp_KeyInsApp≔wp_origin"
    global wp_KeyInsApp=wp_origin
    $ 340 "wp_KeyInsApp[0] = -0.1835 + 0.001"
    wp_KeyInsApp[0] = -0.1835 + 0.001
    $ 341 "wp_KeyInsApp[1] = 0.1105 - 0.003"
    wp_KeyInsApp[1] = 0.1105 - 0.003
    $ 342 "wp_KeyInsApp[5] = 0"
    wp_KeyInsApp[5] = 0
    $ 343 "MoveL"
    $ 344 "wp_KeyInsApp" "breakAfter"
    movel(pose_trans(Fearure_2_2P_Of, wp_KeyInsApp), a=1.2, v=0.25)
    $ 345 "wp_KeyInsert≔wp_KeyInsApp"
    global wp_KeyInsert=wp_KeyInsApp
    $ 346 "wp_KeyInsert[2] = 0.111"
    wp_KeyInsert[2] = 0.111
    $ 347 "MoveL"
    $ 348 "wp_KeyInsert" "breakAfter"
    movel(pose_trans(Fearure_2_2P_Of, wp_KeyInsert), a=1.2, v=0.25)
    # begin: URCap Program Node
    #   Source: Robotiq_Copilot, 1.22.1.14215, Robotiq Inc.
    #   Type: Insertion
    $ 349 "Insertion"
    rq_ft_sensor_disconnected_check()
    # begin: URCap Program Node
    #   Source: Robotiq_Copilot, 1.22.1.14215, Robotiq Inc.
    #   Type: Zero FT Sensor
    $ 350 "Zero FT Sensor" "noBreak"
    rq_ft_sensor_disconnected_check()
    rq_zero_sensor()
    # end: URCap Program Node
    # begin: URCap Program Node
    #   Source: Robotiq_Copilot, 1.22.1.14215, Robotiq Inc.
    #   Type: Linear
    $ 351 "Linear" "noBreak"
    rq_ft_sensor_disconnected_check()
    surface_found = rq_linear_search_urcap("Z+", 10.000, 0.020, 0.030, 1)
    # begin: URCap Program Node
    #   Source: Robotiq_Copilot, 1.22.1.14215, Robotiq Inc.
    #   Type: On error
    $ 352 "On error" "noBreak"
    if not(surface_found):
      $ 353 "'Sequence if maximum distance is reached'" "noBreak"
      # 'Sequence if maximum distance is reached'
      $ 354 "Halt" "noBreak"
      halt
    end
    # end: URCap Program Node
    # end: URCap Program Node
    # end: URCap Program Node
    $ 355 "KeyFeature = get_actual_tcp_pose()"
    KeyFeature =  get_actual_tcp_pose ()
    $ 356 "wp_KeyOrigin[5] = d2r(60)"
    wp_KeyOrigin[5] = d2r(60)
    $ 357 "MoveL"
    $ 358 "wp_KeyOrigin" "breakAfter"
    movel(pose_trans(KeyFeature, wp_KeyOrigin), a=1.2, v=0.1)
    $ 359 "wp_KeyOrigin[5] = 0"
    wp_KeyOrigin[5] = 0
    $ 360 "MoveL"
    $ 361 "wp_KeyOrigin" "breakAfter"
    movel(pose_trans(KeyFeature, wp_KeyOrigin), a=1.2, v=0.1)
    # begin: URCap Program Node
    #   Source: Robotiq_Grippers, 1.8.8.13523, Robotiq Inc.
    #   Type: Gripper
    $ 362 "Gripper Move60% (1)"
    if not(gripper_connected[0]):
      popup("Gripper 1 must be connected to run this program.", "No connection", False, True, True)
    end
    if not(rq_is_gripper_activated("1")):
      popup("Gripper 1 is not activated. Go to Installation tab > Gripper to activate it and run the program again.", "Not activated", False, True, True)
    end
    rq_set_pos_spd_for(153, 0, 0, "1")
    rq_wait_pos_spe_for_request(153, 0, 0, "1")
    rq_go_to("1")
    rq_wait("1")
    # end: URCap Program Node
    $ 363 "wp_KeyInsRet≔wp_KeyInsert"
    global wp_KeyInsRet=wp_KeyInsert
    $ 364 "wp_KeyInsRet[2] = wp_KeyInsRet[2] - 0.111"
    wp_KeyInsRet[2] = wp_KeyInsRet[2] - 0.111
    $ 365 "MoveL"
    $ 366 "wp_KeyInsRet" "breakAfter"
    movel(pose_trans(Fearure_2_2P_Of, wp_KeyInsRet), a=1.2, v=0.25)
    # begin: URCap Program Node
    #   Source: Robotiq_Grippers, 1.8.8.13523, Robotiq Inc.
    #   Type: Gripper
    $ 367 "Gripper Close (1)"
    if not(gripper_connected[0]):
      popup("Gripper 1 must be connected to run this program.", "No connection", False, True, True)
    end
    if not(rq_is_gripper_activated("1")):
      popup("Gripper 1 is not activated. Go to Installation tab > Gripper to activate it and run the program again.", "Not activated", False, True, True)
    end
    rq_set_pos_spd_for(255, 0, 0, "1")
    rq_wait_pos_spe_for_request(255, 0, 0, "1")
    rq_go_to("1")
    rq_wait("1")
    # end: URCap Program Node
  end
  def KeyExtraction():
    $ 368 "KeyExtraction" "noBreak"
    $ 369 "wp_KeyExtApp≔wp_origin"
    global wp_KeyExtApp=wp_origin
    $ 370 "wp_KeyExtApp[0] = wp_KeyExtApp[0] - 0.1820"
    wp_KeyExtApp[0] = wp_KeyExtApp[0] - 0.1820
    $ 371 "wp_KeyExtApp[1] = wp_KeyExtApp[1] + 0.0450"
    wp_KeyExtApp[1] = wp_KeyExtApp[1] + 0.0450
    $ 372 "wp_KeyExtApp[5] = wp_KeyExtApp[5] - 1.571"
    wp_KeyExtApp[5] = wp_KeyExtApp[5] - 1.571
    $ 373 "MoveL"
    $ 374 "wp_KeyExtApp" "breakAfter"
    movel(pose_trans(Fearure_2_2P_Of, wp_KeyExtApp), a=1.2, v=0.25)
    # begin: URCap Program Node
    #   Source: Robotiq_Grippers, 1.8.8.13523, Robotiq Inc.
    #   Type: Gripper
    $ 375 "Gripper Move60% (1)"
    if not(gripper_connected[0]):
      popup("Gripper 1 must be connected to run this program.", "No connection", False, True, True)
    end
    if not(rq_is_gripper_activated("1")):
      popup("Gripper 1 is not activated. Go to Installation tab > Gripper to activate it and run the program again.", "Not activated", False, True, True)
    end
    rq_set_pos_spd_for(153, 0, 0, "1")
    rq_wait_pos_spe_for_request(153, 0, 0, "1")
    rq_go_to("1")
    rq_wait("1")
    # end: URCap Program Node
    $ 376 "wp_KeyExtact≔wp_KeyExtApp"
    global wp_KeyExtact=wp_KeyExtApp
    $ 377 "wp_KeyExtact[2] = wp_KeyExtact[2] + 0.145"
    wp_KeyExtact[2] = wp_KeyExtact[2] + 0.145
    $ 378 "MoveL"
    $ 379 "wp_KeyExtact" "breakAfter"
    movel(pose_trans(Fearure_2_2P_Of, wp_KeyExtact), a=1.2, v=0.25)
    # begin: URCap Program Node
    #   Source: Robotiq_Grippers, 1.8.8.13523, Robotiq Inc.
    #   Type: Gripper
    $ 380 "Gripper Close (1)"
    if not(gripper_connected[0]):
      popup("Gripper 1 must be connected to run this program.", "No connection", False, True, True)
    end
    if not(rq_is_gripper_activated("1")):
      popup("Gripper 1 is not activated. Go to Installation tab > Gripper to activate it and run the program again.", "Not activated", False, True, True)
    end
    rq_set_pos_spd_for(255, 0, 0, "1")
    rq_wait_pos_spe_for_request(255, 0, 0, "1")
    rq_go_to("1")
    rq_wait("1")
    # end: URCap Program Node
    $ 381 "wp_KeyExtRet≔wp_KeyExtact"
    global wp_KeyExtRet=wp_KeyExtact
    $ 382 "wp_KeyExtRet[2] = wp_KeyExtRet[2] - 0.145"
    wp_KeyExtRet[2] = wp_KeyExtRet[2] - 0.145
    $ 383 "MoveL"
    $ 384 "wp_KeyExtRet" "breakAfter"
    movel(pose_trans(Fearure_2_2P_Of, wp_KeyExtRet), a=1.2, v=0.25)
    $ 385 "wp_KeyExtRet[5] = 0"
    wp_KeyExtRet[5] = 0
    $ 386 "MoveL"
    $ 387 "wp_KeyExtRet" "breakAfter"
    movel(pose_trans(Fearure_2_2P_Of, wp_KeyExtRet), a=1.2, v=0.25)
  end
  def PressRedButton():
    $ 388 "PressRedButton" "noBreak"
    $ 389 "wp_RedButApp≔wp_origin"
    global wp_RedButApp=wp_origin
    $ 390 "wp_RedButApp[0] = wp_RedButApp[0] - 0.0555"
    wp_RedButApp[0] = wp_RedButApp[0] - 0.0555
    $ 391 "wp_RedButApp[1] = wp_RedButApp[1] + 0.03"
    wp_RedButApp[1] = wp_RedButApp[1] + 0.03
    $ 392 "MoveL"
    $ 393 "wp_RedButApp" "breakAfter"
    movel(pose_trans(Feature_1, wp_RedButApp), a=1.2, v=0.25)
    $ 394 "Popup"
    popup(str_cat("",wp_RedButApp), "Message", False, False, blocking=True)
    $ 395 "wp_RedButPress≔wp_RedButApp"
    global wp_RedButPress=wp_RedButApp
    $ 396 "wp_RedButPress[2] = wp_RedButPress[2] + 0.125"
    wp_RedButPress[2] = wp_RedButPress[2] + 0.125
    $ 397 "MoveL"
    $ 398 "wp_RedButPress" "breakAfter"
    movel(pose_trans(Feature_1, wp_RedButPress), a=1.2, v=0.25)
    # begin: URCap Program Node
    #   Source: Robotiq_Copilot, 1.22.1.14215, Robotiq Inc.
    #   Type: Find Surface
    $ 399 "Find Surface"
    rq_ft_sensor_disconnected_check()
    rq_zero_sensor()
    sleep(0.1)
    surface_found = rq_linear_search_urcap("Z+", 5.000, 0.030000, 0.010000, 1)
    storevar.setvariablepose("rq_findSurface_e81abd46-3173-4f05-b6bf-f6cecaf39f2c_exitPosition", get_actual_tcp_pose())
    $ 400 "'Add Stop conditions from the Find Surface node'" "noBreak"
    # 'Add Stop conditions from the Find Surface node'
    # begin: URCap Program Node
    #   Source: Robotiq_Copilot, 1.22.1.14215, Robotiq Inc.
    #   Type: If surface found
    $ 401 "If surface found" "noBreak"
    if (surface_found):
      $ 402 "'Sequence if force threshold is reached'" "noBreak"
      # 'Sequence if force threshold is reached'
    end
    # end: URCap Program Node
    # end: URCap Program Node
    $ 403 "wp_RedButRet≔wp_RedButApp"
    global wp_RedButRet=wp_RedButApp
    $ 404 "MoveL"
    $ 405 "wp_RedButRet" "breakAfter"
    movel(pose_trans(Feature_1, wp_RedButRet), a=1.2, v=0.25)
  end
  def PressBlueButton():
    $ 406 "PressBlueButton" "noBreak"
    $ 407 "wp_BluButApp≔wp_origin"
    global wp_BluButApp=wp_origin
    $ 408 "wp_BluButApp[0] = wp_BluButApp[0] - 0.0415"
    wp_BluButApp[0] = wp_BluButApp[0] - 0.0415
    $ 409 "wp_BluButApp[1] = wp_BluButApp[1] + 0.032"
    wp_BluButApp[1] = wp_BluButApp[1] + 0.032
    $ 410 "MoveL"
    $ 411 "wp_BluButApp" "breakAfter"
    movel(pose_trans(Fearure_2_2P_Of, wp_BluButApp), a=1.2, v=0.25)
    $ 412 "wp_BluButPress≔wp_BluButApp"
    global wp_BluButPress=wp_BluButApp
    $ 413 "wp_BluButPress[2] = wp_BluButPress[2] + 0.145"
    wp_BluButPress[2] = wp_BluButPress[2] + 0.145
    $ 414 "MoveL"
    $ 415 "wp_BluButPress" "breakAfter"
    movel(pose_trans(Fearure_2_2P_Of, wp_BluButPress), a=1.2, v=0.25)
    # begin: URCap Program Node
    #   Source: Robotiq_Copilot, 1.22.1.14215, Robotiq Inc.
    #   Type: Find Surface
    $ 416 "Find Surface"
    rq_ft_sensor_disconnected_check()
    rq_zero_sensor()
    sleep(0.1)
    surface_found = rq_linear_search_urcap("Z+", 5.000, 0.030000, 0.010000, 1)
    storevar.setvariablepose("rq_findSurface_1e150698-4c1d-45b1-ae22-50b9cb529eac_exitPosition", get_actual_tcp_pose())
    $ 417 "'Add Stop conditions from the Find Surface node'" "noBreak"
    # 'Add Stop conditions from the Find Surface node'
    # end: URCap Program Node
    $ 418 "wp_BluButRet≔wp_BluButApp"
    global wp_BluButRet=wp_BluButApp
    $ 419 "MoveL"
    $ 420 "wp_BluButRet" "breakAfter"
    movel(pose_trans(Fearure_2_2P_Of, wp_BluButRet), a=1.2, v=0.25)
  end
  def FindCorner():
    $ 421 "FindCorner" "noBreak"
    $ 422 "wp_CornerX≔wp_origin"
    global wp_CornerX=wp_origin
    $ 423 "wp_CornerX[0] = 0.15"
    wp_CornerX[0] = 0.15
    $ 424 "wp_CornerX[5] = 1.571"
    wp_CornerX[5] = 1.571
    $ 425 "MoveL"
    $ 426 "wp_CornerX" "breakAfter"
    movel(pose_trans(Feature_1, wp_CornerX), a=1.2, v=0.5)
    $ 427 "wp_CornerX[2] = 0.18"
    wp_CornerX[2] = 0.18
    $ 428 "MoveL"
    $ 429 "wp_CornerX" "breakAfter"
    movel(pose_trans(Feature_1, wp_CornerX), a=1.2, v=0.25)
    # begin: URCap Program Node
    #   Source: Robotiq_Copilot, 1.22.1.14215, Robotiq Inc.
    #   Type: Find Surface
    $ 430 "Find Surface"
    rq_ft_sensor_disconnected_check()
    rq_zero_sensor()
    sleep(0.1)
    surface_found = rq_linear_search_urcap("Y+", 10.000, 0.030000, 0.030000, 1)
    storevar.setvariablepose("rq_findSurface_b548205b-d40e-4156-b2c2-13eb7d9c5499_exitPosition", get_actual_tcp_pose())
    $ 431 "'Add Stop conditions from the Find Surface node'" "noBreak"
    # 'Add Stop conditions from the Find Surface node'
    # begin: URCap Program Node
    #   Source: Robotiq_Copilot, 1.22.1.14215, Robotiq Inc.
    #   Type: If surface found
    $ 432 "If surface found" "noBreak"
    if (surface_found):
      $ 433 "'Sequence if force threshold is reached'" "noBreak"
      # 'Sequence if force threshold is reached'
      $ 434 "Found_X_Base≔get_actual_tcp_pose()" "noBreak"
      global Found_X_Base= get_actual_tcp_pose ()
      $ 435 "Script: x_dist.script" "noBreak"
      wp_CornerOrigin[0] = sqrt(pow((wp_Center[0] - Found_X_Base[0]), 2) + pow((wp_Center[1] - Found_X_Base[1]), 2))
    end
    # end: URCap Program Node
    # end: URCap Program Node
    $ 437 "wp_CornerX[0] = wp_CornerX[0] + 0.02"
    wp_CornerX[0] = wp_CornerX[0] + 0.02
    $ 438 "MoveL"
    $ 439 "wp_CornerX" "breakAfter"
    movel(pose_trans(Feature_1, wp_CornerX), a=1.2, v=0.25)
    $ 440 "wp_CornerY≔wp_CornerX"
    global wp_CornerY=wp_CornerX
    $ 441 "wp_CornerY[1] =-0.10"
    wp_CornerY[1] =-0.10
    $ 442 "MoveL"
    $ 443 "wp_CornerY" "breakAfter"
    movel(pose_trans(Feature_1, wp_CornerY), a=1.2, v=0.25)
    $ 444 "wp_CornerY[5] = 0"
    wp_CornerY[5] = 0
    $ 445 "MoveL"
    $ 446 "wp_CornerY" "breakAfter"
    movel(pose_trans(Feature_1, wp_CornerY), a=1.2, v=0.5)
    $ 447 "wp_CornerY[0] = 0.05"
    wp_CornerY[0] = 0.05
    $ 448 "MoveL"
    $ 449 "wp_CornerY" "breakAfter"
    movel(pose_trans(Feature_1, wp_CornerY), a=1.2, v=0.25)
    # begin: URCap Program Node
    #   Source: Robotiq_Copilot, 1.22.1.14215, Robotiq Inc.
    #   Type: Find Surface
    $ 450 "Find Surface"
    rq_ft_sensor_disconnected_check()
    rq_zero_sensor()
    sleep(0.1)
    surface_found = rq_linear_search_urcap("Y+", 10.000, 0.030000, 0.040000, 1)
    storevar.setvariablepose("rq_findSurface_f454347d-3177-404d-a22f-0a3a44de9ccc_exitPosition", get_actual_tcp_pose())
    $ 451 "'Add Stop conditions from the Find Surface node'" "noBreak"
    # 'Add Stop conditions from the Find Surface node'
    # begin: URCap Program Node
    #   Source: Robotiq_Copilot, 1.22.1.14215, Robotiq Inc.
    #   Type: If surface found
    $ 452 "If surface found" "noBreak"
    if (surface_found):
      $ 453 "'Sequence if force threshold is reached'" "noBreak"
      # 'Sequence if force threshold is reached'
      $ 454 "Found_Y_Base≔get_actual_tcp_pose()" "noBreak"
      global Found_Y_Base= get_actual_tcp_pose ()
      $ 455 "Script: y_dist.script" "noBreak"
      wp_CornerOrigin[1] = sqrt(pow((wp_Center[0] - Found_Y_Base[0]), 2) + pow((wp_Center[1] - Found_Y_Base[1]), 2))
    end
    # end: URCap Program Node
    # end: URCap Program Node
    $ 457 "wp_CornerY[1] =wp_CornerY[1] - 0.02"
    wp_CornerY[1] =wp_CornerY[1] - 0.02
    $ 458 "MoveL"
    $ 459 "wp_CornerY" "breakAfter"
    movel(pose_trans(Feature_1, wp_CornerY), a=1.2, v=0.25)
    $ 460 "wp_CornerY[2] = 0"
    wp_CornerY[2] = 0
    $ 461 "MoveL"
    $ 462 "wp_CornerY" "breakAfter"
    movel(pose_trans(Feature_1, wp_CornerY), a=1.2, v=0.25)
    $ 463 "Script: without_TCP_offset_dist.script"
    wp_CornerOrigin[0] = wp_CornerOrigin[0] - 0.01
    wp_CornerOrigin[1] = wp_CornerOrigin[1] - 0.01 - 0.0122722
    wp_CornerOrigin[1] = -(wp_CornerOrigin[1])
    wp_CornerOrigin[2] = 0
    $ 464 "MoveL"
    $ 465 "wp_CornerOrigin" "breakAfter"
    movel(pose_trans(Feature_1, wp_CornerOrigin), a=1.2, v=0.25)
    $ 466 "Fearure_2_2P_Of≔get_actual_tcp_pose()"
    global Fearure_2_2P_Of= get_actual_tcp_pose ()
  end
  while (True):
    $ 1 "Robot Program"
    $ 2 "wp_origin≔p[0,0,0,0,0,0]"
    global wp_origin=p[0,0,0,0,0,0]
    $ 3 "wp_KeyOrigin≔p[0,0,0,0,0,0]"
    global wp_KeyOrigin=p[0,0,0,0,0,0]
    $ 4 "wp_CornerOrigin≔p[0,0,0,0,0,0]"
    global wp_CornerOrigin=p[0,0,0,0,0,0]
    # begin: URCap Program Node
    #   Source: Robotiq_Wrist_Camera, 1.11.3.13312, Robotiq Inc.
    #   Type: Cam Locate
    $ 5 "Cam Locate"

    ###########################################
    #######VisionLocate node start########

    f=[0,0.0,0.0,0.0,0.0,0.0,0.0,0]
    object_location=p[0.0,0.0,0.0,0.0,0.0,0.0]
    feature_pose_to_restore_57583 = Calib_4_21May22
    movej([3.910038948059082, -1.5112207571612757, 1.4191160202026367, -0.9934843222247522, -1.6695707480060022, 2.984921932220459])
    # Offset in translation only.
    snapshot_position_offset[3] = 0
    snapshot_position_offset[4] = 0
    snapshot_position_offset[5] = 0
    T_camera_in_flange = p[0, 0, 0, 0, 0, 0] # enlever une fois que l'enseignement du modele sera fait en faisant un movetool avec la pose de la camera dans le repere de la flange. Pour l'instant, on suppose que la camera est situee directement sur la flange.
    tool_57583 = get_T_in_base_from_flange(T_camera_in_flange)
    tool_57583 = pose_sub(tool_57583, snapshot_position_offset)
    snapshot_position = p[0.259014, 0.395272, 0.43384, -0.881995, -2.78157, 0.703037]
    textmsg("expected snapshot position : ", snapshot_position)
    diff = pose_sub(tool_57583, snapshot_position)
    textmsg("diff = ", diff)
    is_at_snapshot_position = norm([diff[0], diff[1], diff[2]]) < 0.002
    is_at_snapshot_position = is_at_snapshot_position and (norm([diff[3], diff[4], diff[5]]) < 0.005)
    textmsg("is_at_snapshot_position = ", is_at_snapshot_position)
    is_snapshot_position_offset = norm(snapshot_position_offset) != 0
    is_at_snapshot_position = is_at_snapshot_position or ignore_snapshot_position
    if not(is_at_snapshot_position):
      popup("Robot is not at Snapshot Position. Add Move instruction to Snapshot Position before Camera Locate node.. Error code: [UCC-8]", warning = False, error = True)
      halt
    end
    f_57583 = xmlrpc_server.findmodel("contextName-57583", tool_57583[0], tool_57583[1], tool_57583[2], tool_57583[3], tool_57583[4], tool_57583[5])
    cam_locate_monitor.setFindModelResult("57583", f_57583)
    canSaveImage = True
    logging_service.publish("FIND_MODEL", f_57583)
    cam_locate_monitor.setCurrentObjectIndex("57583", 0)
    # begin: URCap Program Node
    #   Source: Robotiq_Wrist_Camera, 1.11.3.13312, Robotiq Inc.
    #   Type: Cam Locate Loop
    $ 6 "For object(s) found" "noBreak"
    object_teaching_location_57583 = p[0.2807841967859106, 0.4069757524477864, 0.0014019947306735297, 0.9500904533862067, 2.9785757158511865, 0.006377021049627138]
    feature_teaching_location_57583 = p[0.2807841967859106, 0.4069757524477864, 0.0014019947306735297, 0.9545570299136694, 2.9771536638141938, 0.006412541394240223]
    while (not cam_locate_monitor.isCaptureNeeded("57583")):
      poseAsArray = cam_locate_monitor.getCurrentObjectPoseAsArray("57583")
      current_object_location_57583 = p[poseAsArray[0], poseAsArray[1], poseAsArray[2], poseAsArray[3], poseAsArray[4], poseAsArray[5]]
      object_location = current_object_location_57583
      f[0] = cam_locate_monitor.getNumberOfObjectsFound("57583")
      f[1] = object_location[0]
      f[2] = object_location[1]
      f[3] = object_location[2]
      f[4] = object_location[3]
      f[5] = object_location[4]
      f[6] = object_location[5]
      f[7] = cam_locate_monitor.getCurrentObjectDetectionScore("57583")
      textmsg("current_object_location = ", current_object_location_57583)
      if (norm(snapshot_position_offset) != 0):
        current_object_location_57583 = pose_add(current_object_location_57583, snapshot_position_offset)
        textmsg("current_object_location after snapshot position offset = ", current_object_location_57583)
      end
      Calib_4_21May22 = pose_trans(current_object_location_57583, pose_trans(pose_inv(object_teaching_location_57583), feature_teaching_location_57583))
      $ 7 "target_pose≔object_location" "noBreak"
      global target_pose=object_location
      # begin: URCap Program Node
      #   Source: Robotiq_Grippers, 1.8.8.13523, Robotiq Inc.
      #   Type: Gripper Activate
      $ 8 "Gripper Activate" "noBreak"

      kill rq_gripper_communication_thread
      rq_gripper_communication_thread_started = False
      rq_close_gripper_socket("1")
      rq_close_gripper_socket("2")
      rq_close_gripper_socket("3")
      rq_close_gripper_socket("4")

      rq_init_comm_if_connected(9, "1")
      rq_init_comm_if_connected(2, "2")
      rq_init_comm_if_connected(3, "3")
      rq_init_comm_if_connected(4, "4")
      rq_print_connected_grippers()
      rq_gripper_communication_thread = run rq_gripper_communication()

      while(not rq_gripper_communication_thread_started):
          sleep(0.008)
      end

      rq_set_max_current_for_all_grippers()

      reset_and_activate = False

      rq_activate_all_grippers(False)
      # end: URCap Program Node
      # begin: URCap Program Node
      #   Source: Robotiq_Grippers, 1.8.8.13523, Robotiq Inc.
      #   Type: Gripper
      $ 9 "Gripper Close (1)" "noBreak"
      if not(gripper_connected[0]):
        popup("Gripper 1 must be connected to run this program.", "No connection", False, True, True)
      end
      if not(rq_is_gripper_activated("1")):
        popup("Gripper 1 is not activated. Go to Installation tab > Gripper to activate it and run the program again.", "Not activated", False, True, True)
      end
      rq_set_pos_spd_for(255, 255, 255, "1")
      rq_wait_pos_spe_for_request(255, 255, 255, "1")
      rq_go_to("1")
      rq_wait("1")
      # end: URCap Program Node
      $ 11 "target_pose[2]=target_pose[2]+0.15" "noBreak"
      target_pose[2]=target_pose[2]+0.15
      $ 12 "MoveL" "noBreak"
      $ 13 "target_pose" "noBreak"
      movel(pose_trans(p[0.0,0.0,0.0,0.0,0.0,0.0], target_pose), a=1.2, v=0.25)
      $ 14 "wp_Center≔get_actual_tcp_pose()" "noBreak"
      global wp_Center= get_actual_tcp_pose ()
      $ 16 "Feature_1≔target_pose" "noBreak"
      global Feature_1=target_pose
      $ 17 "Call FindCorner" "noBreak"
      FindCorner()
      $ 34 "Call PickPlaceCoinBattery" "noBreak"
      PickPlaceCoinBattery()
      $ 36 "Halt" "noBreak"
      halt
      cam_locate_monitor.incrementIndex("57583")
    end
    # end: URCap Program Node
    # begin: URCap Program Node
    #   Source: Robotiq_Wrist_Camera, 1.11.3.13312, Robotiq Inc.
    #   Type: If no object found in Camera Locate
    $ 37 "If no object found" "noBreak"
    if (not cam_locate_monitor.hasFoundObjects("57583")):
      f[0] = 0
      $ 38 "'Optional'" "noBreak"
      # 'Optional'
    end
    # end: URCap Program Node
    # Restore feature pose
    Calib_4_21May22 = feature_pose_to_restore_57583

    #######VisionLocate node end########
    ###########################################

    # end: URCap Program Node
  end
end
